// TIA Portal V18 export
DATA_BLOCK "PROFINET_NODES_ALARM"   // DB10
{ S7_Optimized_Access := 'TRUE' }
VERSION : 0.1
// stored: AutoNumber true, DBAccessibleFromOPCUA true, DBAccessibleFromWebserver true
   VAR
      AlwaysFALSE : Bool;
      AlwaysTRUE : Bool;
      "No Operation" : Bool;
      "n0006-mc1-cc1-k66201 192.168.50.6" : Bool;
      "n0005-ms1-cc1-k65001 192.168.50.5" : Bool;
      "n0012-pc1-cc1-k65001 192.168.50.12" : Bool;
      "n0031-sm72-xns1 192.168.50.31" : Bool;
      "n0005-ms2-cc1-k65001 192.168.51.5" : Bool;
      "n0012-pc2-cc1-k65001 192.168.51.12" : Bool;
      "n0031-sm73-xns1 192.168.51.31" : Bool;
   END_VAR
BEGIN
END_DATA_BLOCK
